Yaskawa INFORM job: 80_180.JBI

/JOB
//NAME 80_180
///FOLDERNAME OBROTNIK
//POS
///NPOS 0,0,1,0,0,0
///TOOL 0
///POSTYPE PULSE
///PULSE
EC00000=709473,1112952
//INST
///DATE 2023/11/07 19:19
///ATTR SC,RW,RJ
////FRAME ROBOT
///GROUP1 ST1
NOP
MOVJ EC00000 VJ=100.00
END
